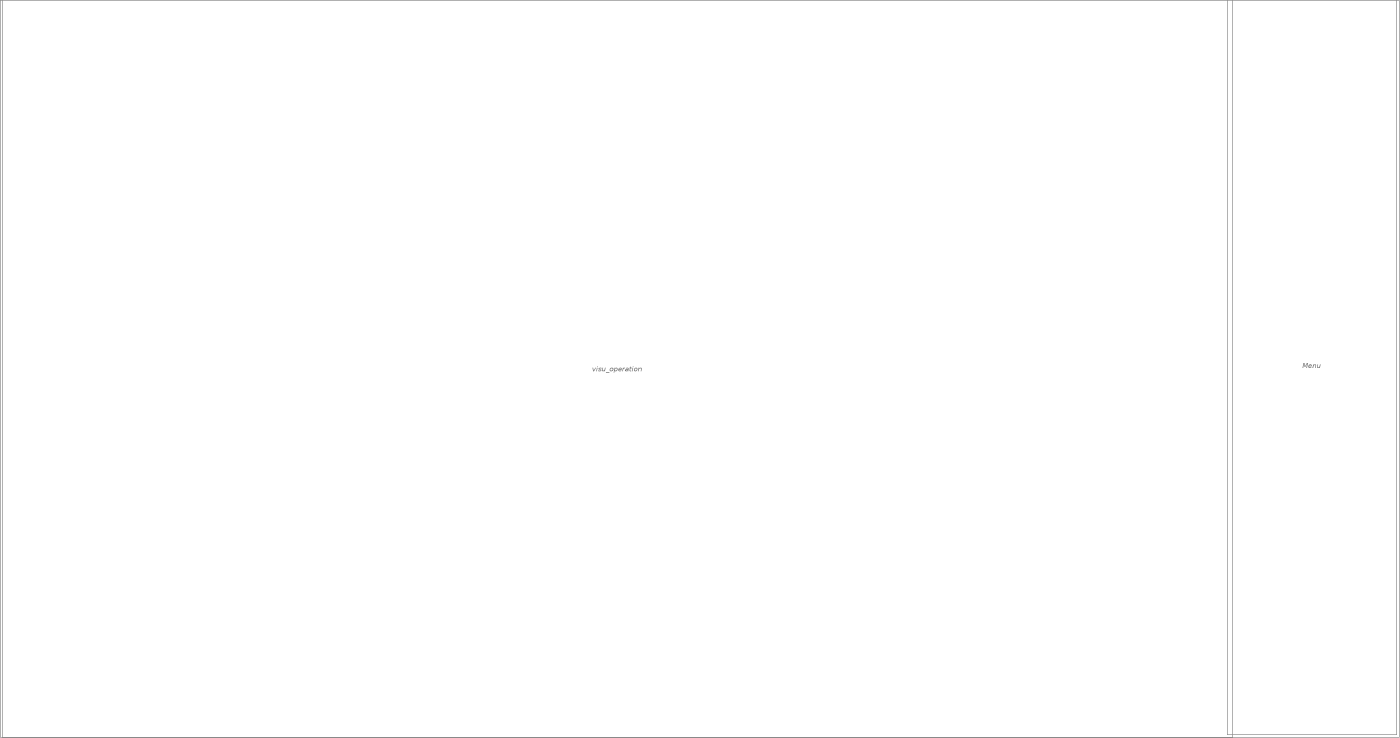
VISUALIZATION visu_manual  // 2048x1080
    Frame (3,0 1800x1080), frame switch variable: G_HMI.iMainFrame
        shows visu_operation()
        shows v_alarm()
        shows visu_loading()
        shows visu_working1()
        shows visu_working2()
        shows visu_2sys()
    Frame (1795,-5 248x1080), frame switch variable: G_HMI.iMainFrame
        shows Menu()
        shows visu_working()
        shows v_IO_fixtureClamp()
        shows visu_buffer()
        shows visu_loading()
        shows v_alarm()
END_VISUALIZATION

(* stored: Version 1.1.0.1, ProductVersion 3.1.4024.12
   Visu visu_manual: Id {27f18664-69ba-41bf-9a81-29f5cd36101a} *)
